Omron CX-Programmer project NewProject (CX-Programmer 9.73)

# PLC NewPLC1: CJ2M CPU11

## Global symbols (name address type ; comment)
0.00 BOOL  ; STOP
0.01 BOOL  ; START
0.02 BOOL  ; SENSOR MERAH
0.03 BOOL  ; SENSOR LABEL
0.04 BOOL  ; SENSOR BIRU
0.05 BOOL  ; EMERGENCY STOP
100.00 BOOL  ; MOTOR CONVEYOR
100.01 BOOL  ; Pneumatic MERAH
100.02 BOOL  ; Pneumatic BIRU
100.03 BOOL  ; Lampu Hijau
100.04 BOOL  ; Lampu Merah
1.01 BOOL  ; CONVEYOR
T0000 BOOL  ; TIMER Pneumatic MERAH
T0001 BOOL  ; TIMER Pneumatic BIRU

## Program NewProgram1 (cyclic task 0)
Local symbols
T BOOL

### Section Section1

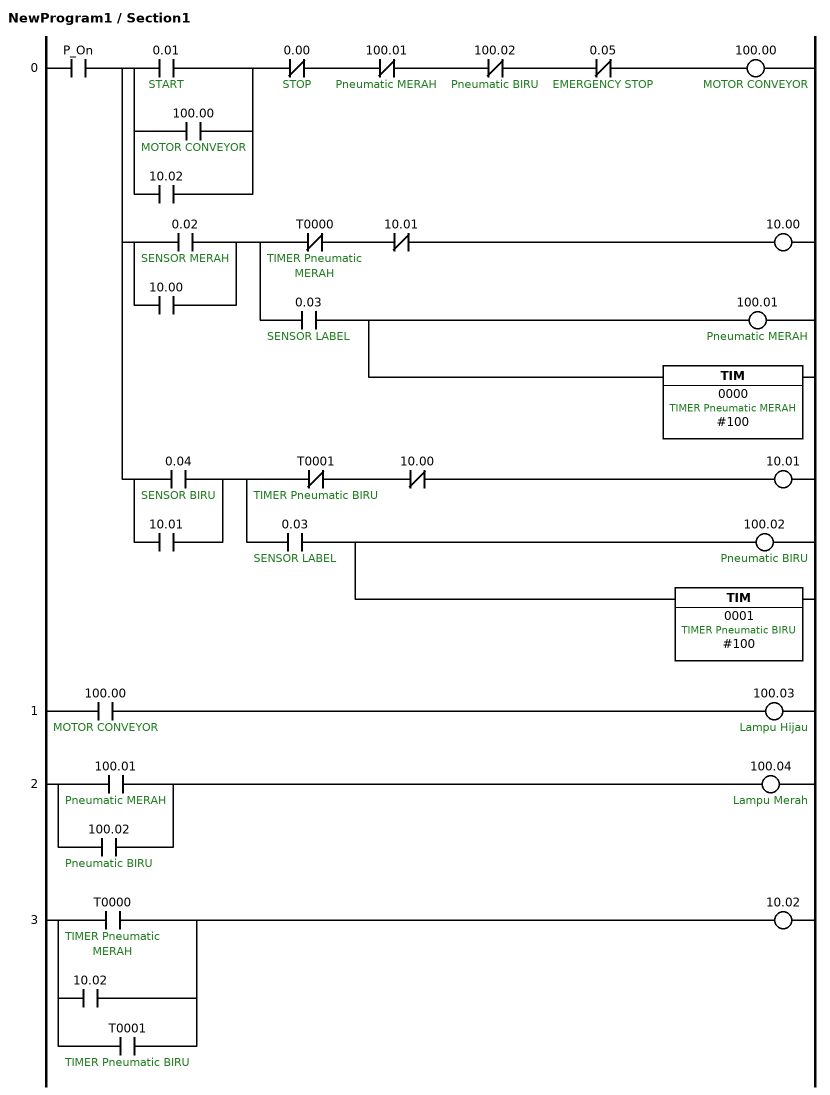
; rung 0
LD P_On
OUT TR0
LD 0.01  ; START
OR 100.00  ; MOTOR CONVEYOR
OR 10.02
ANDLD
ANDNOT 0.00  ; STOP
ANDNOT 100.01  ; Pneumatic MERAH
ANDNOT 100.02  ; Pneumatic BIRU
ANDNOT 0.05  ; EMERGENCY STOP
OUT 100.00  ; MOTOR CONVEYOR
LD TR0
LD 0.02  ; SENSOR MERAH
OR 10.00
ANDLD
OUT TR1
ANDNOT T0000  ; TIMER Pneumatic MERAH
ANDNOT 10.01
OUT 10.00
LD TR1
AND 0.03  ; SENSOR LABEL
OUT 100.01  ; Pneumatic MERAH
TIM 0000 #100  ; TIMER Pneumatic MERAH
LD TR0
LD 0.04  ; SENSOR BIRU
OR 10.01
ANDLD
OUT TR0
ANDNOT T0001  ; TIMER Pneumatic BIRU
ANDNOT 10.00
OUT 10.01
LD TR0
AND 0.03  ; SENSOR LABEL
OUT 100.02  ; Pneumatic BIRU
TIM 0001 #100  ; TIMER Pneumatic BIRU
; rung 1
LD 100.00  ; MOTOR CONVEYOR
OUT 100.03  ; Lampu Hijau
; rung 2
LD 100.01  ; Pneumatic MERAH
OR 100.02  ; Pneumatic BIRU
OUT 100.04  ; Lampu Merah
; rung 3
LD T0000  ; TIMER Pneumatic MERAH
OR 10.02
OR T0001  ; TIMER Pneumatic BIRU
OUT 10.02

### Section END
; rung 0
END(001)